{region '#Template'}
	{attribute 'Version' := '5.0.0.0'}
	{attribute 'Tags' := '"LCID": "1031", "Text": "Gebäudeautomation, Kommunikation, Server, Client, Publisher, Subscriber"'}
	{attribute 'Tags' := '"LCID": "1033", "Text": "Building automation, Communication, Server, Client, Publisher, Subscriber"'}
	{attribute 'Using' := '"Type": "Template", "URI": "Site"'}
	{attribute 'Description' := '"LCID": "1031", "Text": "Server Datenkommunikation"'}
	{attribute 'Description' := '"LCID": "1033", "Text": "Server data communication"'}
{endregion}

FUNCTION_BLOCK FB_BA_AdsComServer
VAR_INPUT
END_VAR
VAR_OUTPUT
END_VAR
VAR_INPUT CONSTANT
	WeatherStation					: FB_BA_RawPublisher;			
	GeneralSettings					: FB_BA_RawPublisher;												
END_VAR
VAR
END_VAR

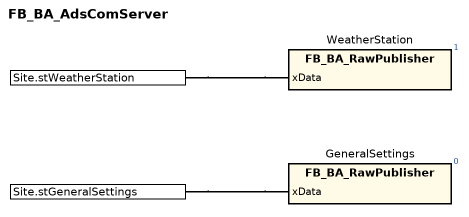
GeneralSettings(xData := Site.stGeneralSettings); // FB_BA_RawPublisher
WeatherStation(xData := Site.stWeatherStation); // FB_BA_RawPublisher

END_FUNCTION_BLOCK

(* stored: Version 1.1.0.1, ProductVersion 3.1.4024.12
   POU FB_BA_AdsComServer: Id {1b1bf36b-f457-49d8-b0b3-98563e0f98b0}, SpecialFunc None *)
